// TIA Portal V16 export
// export: Created 2022-03-28T07:44:07.9426657Z, ExportSetting WithDefaults, DisplayName Totally Integrated Automation Portal, DisplayVersion V16 Update 5, DisplayName TIA Portal Version Control Interface, DisplayVersion V16 Update 2, DisplayName TIA Portal Openness, DisplayVersion V16 Update 5, DisplayName STEP 7 Professional, DisplayVersion V16 Update 5, DisplayName STEP 7 Safety, DisplayVersion V16, DisplayName WinCC Professional, DisplayVersion V16 Update 5
DATA_BLOCK "dbi_fb_01_Cycle"   // DB1
VERSION : 0.1
// stored: AutoNumber false, InstanceOfName fb_01_Cycle, InstanceOfType FB
"fb_01_Cycle"
   // VAR
   //    TON_Delay : Array[1..10] of TON_TIME;
   //    TP_Reset { S7_SetPoint := 'True'} : TP_TIME;
   // END_VAR
BEGIN
END_DATA_BLOCK
